(*			
	RAFALOS
	Rafał Osajda		23.09.2025		TC 4024.66
	Struktura pomocnicza potrzeba do wiazania zmiennych
*)
TYPE ST_BaseHMIComponent_Command_Link :
STRUCT
	stBaseLoggerElement				: ST_BaseHMILoggerElement_View;
	stBaseComponent					: ST_BaseHMIComponent_View;
END_STRUCT
END_TYPE

(* stored: Version 1.1.0.1
   DUT ST_BaseHMIComponent_Command_Link: Id {a40c4165-7f8b-0efc-0bc6-218f72422b6e} *)
